INTERFACE I_State

PROPERTY Description : STRING
GET
END_GET
END_PROPERTY

METHOD DetectedPartSensor1 : BOOL
VAR_INPUT
END_VAR
END_METHOD

METHOD DetectedPartSensor2 : BOOL
VAR_INPUT
END_VAR
END_METHOD

METHOD DetectedWeightSensor : BOOL
VAR_INPUT
END_VAR
END_METHOD

METHOD PressEmergencyStop : BOOL
VAR_INPUT
END_VAR
END_METHOD

METHOD PressStart : BOOL
VAR_INPUT
END_VAR
END_METHOD

METHOD PressStop : BOOL
VAR_INPUT
END_VAR
END_METHOD

METHOD ProcessedWeight : BOOL
VAR_INPUT
END_VAR
END_METHOD

END_INTERFACE

(* stored: Version 1.1.0.1, ProductVersion 3.1.4024.12
   Itf I_State: Id {7077d6f2-af75-4940-9f81-39240c480972}
   Property Description: Id {fccbae2c-8d35-49aa-9486-489996ac39de}
   Get Get: Id {d900df21-e5ef-484e-91f8-86586596cd0e}
   Method DetectedPartSensor1: Id {b7326d1e-3882-4365-a65e-3d2f84738e34}
   Method DetectedPartSensor2: Id {036f2692-c892-4b92-9cde-39234bc3f211}
   Method DetectedWeightSensor: Id {969cf619-fcb0-4e53-91b6-74ce40a43ac2}
   Method PressEmergencyStop: Id {b3e75f9c-9ca4-4351-8c78-7257e7b10cb0}
   Method PressStart: Id {f8e9b630-d84e-490e-991e-88d478b496a3}
   Method PressStop: Id {3d536037-4385-4003-879f-723b14d4144c}
   Method ProcessedWeight: Id {01b8e78e-f948-457d-8004-f458df044f30} *)
